// TIA Portal V16 export
// export: Created 2021-07-12T14:47:19.9612721Z, ExportSetting WithDefaults, DisplayName Totally Integrated Automation Portal, DisplayVersion V16, DisplayName TIA Portal Version Control Interface, DisplayVersion V16, DisplayName TIA Portal Openness, DisplayVersion V16, DisplayName STEP 7 Professional, DisplayVersion V16, DisplayName STEP 7 Safety, DisplayVersion V16, DisplayName WinCC Professional, DisplayVersion V16
TYPE "LSimaHydTO_typeMeasuredValues"
TITLE = LSimaHydTO_typeMeasuredValues
// Measurement results
// stored: IsFailsafeCompliant false
   STRUCT
      forward { S7_SetPoint := 'True'} : "LSimaHydTO_typeVCharMeasured";   // measured values in positive direction
      backward { S7_SetPoint := 'True'} : "LSimaHydTO_typeVCharMeasured";   // measured values in negative direction
   END_STRUCT;
END_TYPE
